RoboDK station: PROYECTO DE MECANIZADO inicial.rdk

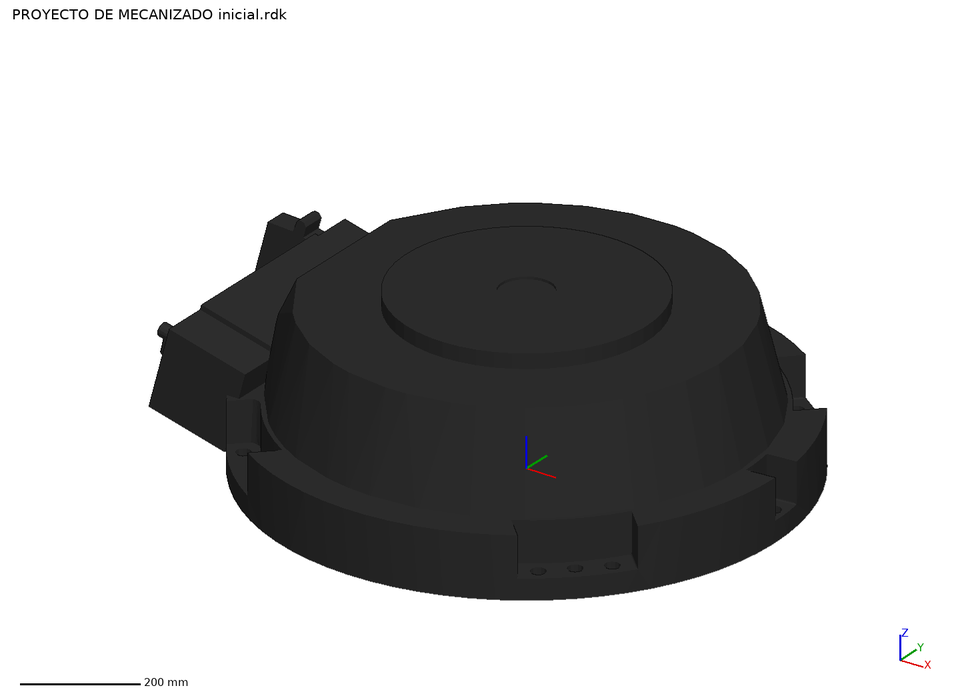
[picture v0: the station drawn from its stored meshes, robots at their saved joint values, targets as dots, program paths as lines]
Station PROYECTO DE MECANIZADO inicial (saved by RoboDK 5.7.5). Poses are relative to the parent item; angles as X-Y-Z fixed-axis rotations.
  - frame ORIGEN at (0, 0, 0) mm
  - frame KUKA KR 200 comp Base at (0, 0, 0) mm
    - robot KUKA KR 200 comp: 6 axes
        joint limits [-185, -142, -120, -350, -120, -350] to [185, 0, 148, 350, 120, 350]; home [0, -90, 90, 0, 0, 0]; saved at [-18.305, -63.639, 118.623, 158.005, 56.991, -167.59]
      - tool Teknomotor ATC710039 Spindle, TCP at (296, 0, 80.3) mm, rotated rx 0 ry 90 rz 0 deg, size 475 x 150 x 192.7 mm
        - object ENDMILL_D16_150 at (0, 0, 0) mm, rotated rx 180 ry 0 rz 0 deg, size 16 x 16 x 150 mm, geometry from ENDMILL_D16_150.IGS
  - frame MECANIZADO at (1500, 0, 250) mm
    - object 500x500x250 at (0, 0, 0) mm, size 500 x 500 x 250 mm, geometry from 500x500x250.STEP
